TYPE ST_Event :
STRUCT
	eEventType		: E_eventType ;	// Verbose:= 0, Info := 1, Warning  := 2,  Error := 3, Critical := 4
	nEventIdentity	: UDINT ;
	strEventText	: STRING(50);
	dtTimeStamp		: DATE_AND_TIME;
END_STRUCT
END_TYPE

(* stored: Version 1.1.0.1, ProductVersion 3.1.4024.15
   DUT ST_Event: Id {57e09a9f-e6db-43be-9332-7969c9378537} *)
